// SIMATIC S7-200 project (STEP 7-Micro/WIN), CPU 222 REL 02.01

SYMBOL_TABLE USER1
NO_BEVANDA       M0.5     // NESSUNA BEVANDA SELEZIONATA
BEV_1            Q0.0     // BEVANDA 1
BEV_2            Q0.1     // BEVANDA 2
BEV_3            Q0.2     // BEVANDA 3
BEV_4            Q0.3     // BEVANDA 4
RESO_M           Q0.4     // RESO MONETA
SEL_BEV_1        I0.0     // SELEZIONE BEVANDA 1
SEL_BEV_2        I0.1     // SELEZIONE BEVANDA 2
SEL_BEV_3        I0.2     // SELEZIONE BEVANDA 3
SEL_BEV_4        I0.3     // SELEZIONE BEVANDA 4
RIT_BEV          I0.4     // RITIRO BEVANDA
MON_ESATTO       I0.5     // RICONOSCIMENTO INSERIMENTO MONETA ESATTO
MON_ERRATO       I0.6     // RICONOSCIMENTO INSERIMENTO MONETA ERRATA
RESO             I0.7     // RESO MONETA
RESTIT_MON       I1.0     // RESTITUZIONE MONETA
END_SYMBOL_TABLE

ORGANIZATION_BLOCK MAIN:OB1
TITLE=DPS 204 DISTRIBUTORE BEVANDE
BEGIN
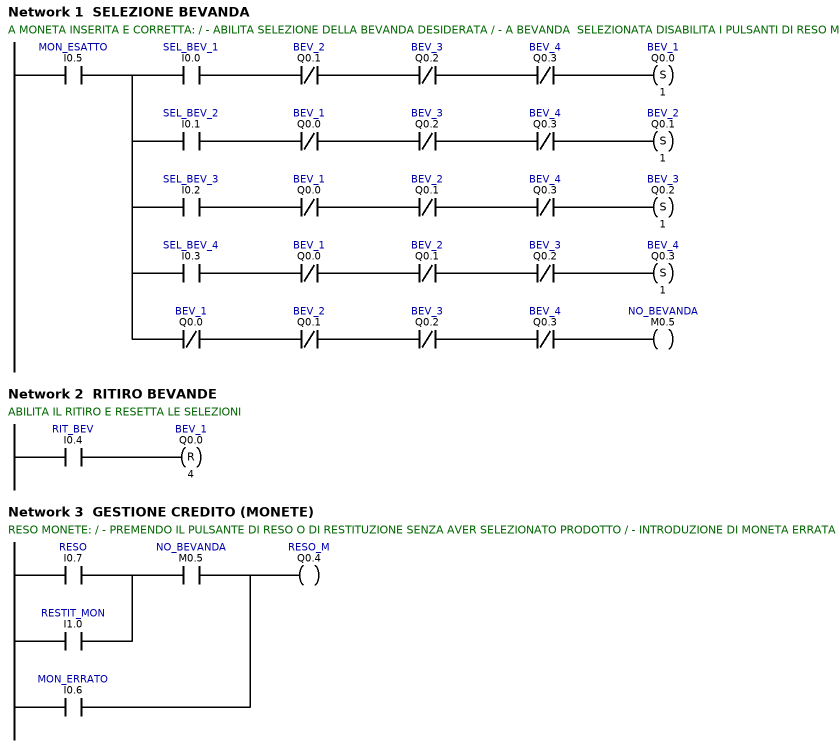
Network 1 // SELEZIONE BEVANDA
// A MONETA INSERITA E CORRETTA:
// - ABILITA SELEZIONE DELLA BEVANDA DESIDERATA
// - A BEVANDA  SELEZIONATA DISABILITA I PULSANTI DI RESO MONETA E RESTITUZIONE MONETA
// 
LD     MON_ESATTO:I0.5
LPS
A      SEL_BEV_1:I0.0
AN     BEV_2:Q0.1
AN     BEV_3:Q0.2
AN     BEV_4:Q0.3
S      BEV_1:Q0.0, 1
LRD
A      SEL_BEV_2:I0.1
AN     BEV_1:Q0.0
AN     BEV_3:Q0.2
AN     BEV_4:Q0.3
S      BEV_2:Q0.1, 1
LRD
A      SEL_BEV_3:I0.2
AN     BEV_1:Q0.0
AN     BEV_2:Q0.1
AN     BEV_4:Q0.3
S      BEV_3:Q0.2, 1
LRD
A      SEL_BEV_4:I0.3
AN     BEV_1:Q0.0
AN     BEV_2:Q0.1
AN     BEV_3:Q0.2
S      BEV_4:Q0.3, 1
LPP
AN     BEV_1:Q0.0
AN     BEV_2:Q0.1
AN     BEV_3:Q0.2
AN     BEV_4:Q0.3
=      NO_BEVANDA:M0.5
Network 2 // RITIRO BEVANDE
// ABILITA IL RITIRO E RESETTA LE SELEZIONI
LD     RIT_BEV:I0.4
R      BEV_1:Q0.0, 4
Network 3 // GESTIONE CREDITO (MONETE)
// RESO MONETE:
// - PREMENDO IL PULSANTE DI RESO O DI RESTITUZIONE SENZA AVER SELEZIONATO PRODOTTO
// - INTRODUZIONE DI MONETA ERRATA
LD     RESO:I0.7
O      RESTIT_MON:I1.0
A      NO_BEVANDA:M0.5
O      MON_ERRATO:I0.6
=      RESO_M:Q0.4
Network 4
// MEND
END_ORGANIZATION_BLOCK
